FUNCTION TryConvert_TIME_TO_BYTE : BOOL
VAR_INPUT
	in : TIME;
	out : REFERENCE TO BYTE;
END_VAR

IF in > DatatypeLimits.MAX_VALUE_OF_TIME_WHICH_CAN_BE_HELD_IN_A_BYTE THEN
	RETURN;
END_IF

out := TIME_TO_BYTE(in);
TryConvert_TIME_TO_BYTE := TRUE;

END_FUNCTION

(* stored: Version 1.1.0.1, ProductVersion 3.1.4024.12
   POU TryConvert_TIME_TO_BYTE: Id {52f5f03b-2e01-43f8-a866-f12294f4f9b2}, SpecialFunc None *)
